(* CODESYS project FsTime_0.1.0.0.library
   Company: FisoThemes
   DefaultNamespace: FsTime
   Version: 0.1.0.0
   Placeholder: FsTime
   Author: Goodwill Mzumala
   Description: A library for time management and manipulation.
   Title: FsTime

Project tree, tasks and I/O mapping:
  libraries: FsCommon, * (FisoThemes); FsError, * (FisoThemes); SysTime, 3.5.9.0 (System); Tc2_Standard, * (Beckhoff Automation GmbH); Tc2_System, * (Beckhoff Automation GmbH); Tc3_Module, * (Beckhoff Automation GmbH)
  DUTs/
    data type E_DayOfWeek
    data type E_Month
    data type E_TimeInstanceKind
    data type T_DayOfMonth
    data type T_DayOfYear
    data type T_Hour
    data type T_Microsecond
    data type T_Millisecond
    data type T_Minute
    data type T_Nanosecond
    data type T_Second
    data type T_Year
  GVLs/
  ITFs/
    Time Instance/
      interface I_ComparableTimesInstance: IsAfter, IsBefore, IsEqualTo
      interface I_EquatableTimesInstance: IsEqualTo
      interface I_TimeInstance: DayOfMonth, DayOfWeek, DayOfYear, EpochMilliseconds, Hour, IsAfter, IsBefore, IsEqualTo, Kind, Millisecond, Minute, Month, Second, ToDate, ToDateTime, ToLocal, ToTimeOfDay, ToUTC, Year
      interface I_TimeInstanceArithmetics
      interface I_TimeInstanceConversions: ToDate, ToDateTime, ToLocal, ToTimeOfDay, ToUTC
      interface I_TimeInstanceProperties: DayOfMonth, DayOfWeek, DayOfYear, EpochMilliseconds, Hour, Kind, Millisecond, Minute, Month, Second, Year
    Time Span/
      interface I_TimeSpan: Day, Hour, Microsecond, Millisecond, Minute, Nanosecond, Second, Tick, ToDays, ToHours, ToMicroseconds, ToMilliseconds, ToMinutes, ToNanoseconds, ToSeconds
      interface I_TimeSpanConversions: ToDays, ToHours, ToMicroseconds, ToMilliseconds, ToMinutes, ToNanoseconds, ToSeconds
      interface I_TimeSpanProperties: Day, Hour, Microsecond, Millisecond, Minute, Nanosecond, Second, Tick
    interface I_IntervalTimer: ElapsedTime, IntervalCount, IntervalTime, IsRunning, Run, SetCallback, Start, Stop
    interface I_Stopwatch: Clear, ElapsedTime, IsRunning, Start, Stop
    interface I_TimeElapsedCallback: OnTimeElapsed
    interface I_Timer: Clear, Duration, ElapsedTime, HasExpired, HasPaused, IsRunning, Pause, Start, Stop, TimeRemaining
    interface I_TimingSource
  POUs/
    function block FB_IntervalTimer [ST]: ElapsedTime, IntervalCount, IntervalTime, IsRunning, Run, SetCallback, Start, Stop
    function block FB_Stopwatch [ST]: Clear, ElapsedTime, IsRunning, Start, Stop
    function block FB_TimeInstance [ST]: DayOfMonth, DayOfWeek, DayOfYear, EpochMilliseconds, FromDate, FromDateTime, FromEpochMilliseconds, FromTime, FromTimeOfDay, Hour, Instance, IsAfter, IsBefore, IsEqualTo, Kind, Millisecond, Minute, Month, Now, Second, ToDate, ToDateTime, ToLocal, ToTimeOfDay, ToUTC, Year
    function block FB_Timer [ST]: Clear, Duration, ElapsedTime, HasExpired, HasPaused, IsRunning, Pause, Start, Stop, TimeRemaining
    function block FB_TimeSpan [ST]: Day, FromShortTime, FromTime, Hour, Microsecond, Millisecond, Minute, Nanosecond, Now, Second, Span, Tick, ToDays, ToHours, ToMicroseconds, ToMilliseconds, ToMinutes, ToNanoseconds, ToSeconds
    program PLAYGROUND [ST]: Example1
  Project Information/
    function F_GetCompany [ST]
    function F_GetTitle [ST]
    function F_GetVersion [ST]
  Version/
    global variables Global_Version
  VISUs/
*)

// DUTs/E_DayOfWeek
// Represents the days of the week.
{attribute 'qualified_only'}
{attribute 'to_string'}
TYPE E_DayOfWeek :
(
	_ := 0, // Uninitialised or default value, representing an undefined day.
	Monday,
	Tuesday,
	Wednesday,
	Thursday,
	Friday,
	Saturday,
	Sunday
) UINT;
END_TYPE

// DUTs/E_Month
// Represents the months of the year.
{attribute 'qualified_only'}
{attribute 'to_string'}
TYPE E_Month :
(
	_ := 0, // Uninitialised or default value, representing an undefined month.
	January,
	February,
	March,
	April,
	May, 
	June, 
	July,
	August,
	September,
	October,
	November,
	December
)UINT;
END_TYPE

// DUTs/E_TimeInstanceKind
{attribute 'qualified_only'}
{attribute 'to_string'}
TYPE E_TimeInstanceKind :
(
	_ := 0, // Uninitialised or default value, indicating an undefined time instance kind.
	UTC,  // The time instance is in Coordinated Universal Time (UTC).
	Local // The time instance is in local time.
);
END_TYPE

// DUTs/T_DayOfMonth
// Represents the day of the current month, with values ranging from 1 to 31, based on the month.
TYPE T_DayOfMonth : UINT(1..31); END_TYPE

// DUTs/T_DayOfYear
// Represents the day of the year, ranging from 1 to 366, where 1 is January 1st,
// and 365 or 366 is December 31st (accounts for leap years).
TYPE T_DayOfYear : UINT(1..366); END_TYPE

// DUTs/T_Hour
// Represents the hours of the current day, based on a 24-hour format, ranging from 0 to 23.
TYPE T_Hour : UINT(0..23); END_TYPE

// DUTs/T_Microsecond
// Represents the microseconds of the current millisecond, ranging from 0 to 999.
TYPE T_Microsecond : UINT(0..999); END_TYPE

// DUTs/T_Millisecond
// Represents the milliseconds of the current second, ranging from 0 to 999.
TYPE T_Millisecond : UINT(0..999); END_TYPE

// DUTs/T_Minute
// Represents the minutes of the current hour, ranging from 0 to 59.
TYPE T_Minute : UINT(0..59); END_TYPE

// DUTs/T_Nanosecond
// Represents the nanoseconds of the current microsecond, ranging from 0 to 999.
TYPE T_Nanosecond : UINT(0..999); END_TYPE

// DUTs/T_Second
// Represents the seconds of the current minute, ranging from 0 to 59.
TYPE T_Second : UINT(0..59); END_TYPE

// DUTs/T_Year
// Represents the year as a four-digit value (e.g., 2024).
TYPE T_Year : UINT; END_TYPE

// Version/Global_Version
{attribute 'TcGenerated'}
{attribute 'no-analysis'}
{attribute 'linkalways'}
// This function has been automatically generated from the project information.
VAR_GLOBAL CONSTANT
	{attribute 'const_non_replaced'}
	stLibVersion_FsTime : ST_LibVersion := (iMajor := 0, iMinor := 1, iBuild := 0, iRevision := 0, nFlags := 0, sVersion := '0.1.0.0');
END_VAR

// ITFs/Time Instance/I_ComparableTimesInstance
// This interface defines operations for comparing time instance objects within a system.
INTERFACE I_ComparableTimesInstance EXTENDS __SYSTEM.IQueryInterface

// Checks if the current time instance is after the specified time instance.
METHOD IsAfter : BOOL // TRUE if the current time instance is after the specified one, FALSE otherwise.
VAR_INPUT
	// The time instance to compare against.
	ipOther : I_TimeInstance;
END_VAR
END_METHOD

// Checks if the current time instance is before the specified time instance.
METHOD IsBefore : BOOL // TRUE if the current time instance is before the specified one, FALSE otherwise.
VAR_INPUT
	// The time instance to compare against.
	ipOther : I_TimeInstance;
END_VAR
END_METHOD

// Checks if the current time instance is equal to the specified time instance.
METHOD IsEqualTo : BOOL // TRUE if the current time instance is equal to the specified, FALSE otherwise.
VAR_INPUT
	// The time instance to compare against.
	ipOther : I_TimeInstance;
END_VAR
END_METHOD

END_INTERFACE

// ITFs/Time Instance/I_TimeInstance
// Interface for a time instance.
INTERFACE I_TimeInstance EXTENDS __SYSTEM.IQueryInterface

// The day of the month extracted from the time instance.
// [get] Returns the day component of the date, with a value ranging from 1 to 31.
PROPERTY DayOfMonth : T_DayOfMonth
GET
END_GET
END_PROPERTY

// The day of the week extracted from the time instance.
// [get] Returns the day as an `E_DayOfWeek` enum or value ranging from 1 (Monday) to 7 (Sunday).
PROPERTY DayOfWeek : E_DayOfWeek
GET
END_GET
END_PROPERTY

// The day of the year extracted from the time instance.
// [get] Returns the day of the year, with a value ranging from 1 to 366.
PROPERTY DayOfYear : T_DayOfYear
GET
END_GET
END_PROPERTY

// The time instance value represented as the number of milliseconds since
// Thursday, 1.1.1970 00:00:00.000 (Unix epoch).
// [get] Returns the time instance value in milliseconds.
PROPERTY EpochMilliseconds : ULINT
GET
END_GET
END_PROPERTY

// The hour of the day extracted from the time instance.
// [get] Returns the hour component of the time, with a value ranging from 0 to 23.
PROPERTY Hour : T_Hour
GET
END_GET
END_PROPERTY

// Checks if the current time instance is after the specified time instance.
METHOD IsAfter : BOOL // TRUE if the current time instance is after the specified one, FALSE otherwise.
VAR_INPUT
	// The time instance to compare against.
	ipOther : I_TimeInstance;
END_VAR
END_METHOD

// Checks if the current time instance is before the specified time instance.
METHOD IsBefore : BOOL // TRUE if the current time instance is before the specified one, FALSE otherwise.
VAR_INPUT
	// The time instance to compare against.
	ipOther : I_TimeInstance;
END_VAR
END_METHOD

// Checks if the current time instance is equal to the specified time instance.
METHOD IsEqualTo : BOOL // TRUE if the current time instance is equal to the specified, FALSE otherwise.
VAR_INPUT
	// The time instance to compare against.
	ipOther : I_TimeInstance;
END_VAR
END_METHOD

// Specifies whether the time instance is in UTC or local time format.
// [get] Returns the time instance type enum as a value.
PROPERTY Kind : E_TimeInstanceKind
GET
END_GET
END_PROPERTY

// The millisecond part of the second extracted from the time instance.
// [get] Returns the millisecond component, with a value ranging from 0 to 999.
PROPERTY Millisecond : T_Millisecond
GET
END_GET
END_PROPERTY

// The minute of the hour extracted from the time instance.
// [get] Returns the minute component, with a value ranging from 0 to 59.
PROPERTY Minute : T_Minute
GET
END_GET
END_PROPERTY

// The month of the year extracted from the time instance.
// [get] Returns the month as an `E_Month` enum or a value ranging from 1 to 12 value.
PROPERTY Month : E_Month
GET
END_GET
END_PROPERTY

// The second of the minute extracted from the time instance.
// [get] Returns the second component, with a value ranging from 0 to 59.
PROPERTY Second : T_Second
GET
END_GET
END_PROPERTY

// Converts the time instance to a date value.
METHOD ToDate : DATE // The date part of the time instance.
VAR_OUTPUT
	// Error code indicating the result of the operation.
	Error : FsError.T_Error;
END_VAR
END_METHOD

// Converts the time instance to a combined date and time value.
METHOD ToDateTime : DT // The combined date and time value as a DT (Date and Time).
VAR_OUTPUT
	// Error code indicating the result of the operation.
	Error : FsError.T_Error;
END_VAR
END_METHOD

// Converts the time instance to local time representation.
METHOD ToLocal : I_TimeInstance // A reference to the current instance.
VAR_OUTPUT
	// Error code indicating the result of the operation.
	Error : FsError.T_Error;
END_VAR
END_METHOD

// Converts the time instance to a time of day  value.
METHOD ToTimeOfDay : TOD // The time of day part of the time instance.
VAR_INPUT
END_VAR
END_METHOD

// Converts the time instance to UTC time representation.
METHOD ToUTC : I_TimeInstance // A reference to the current instance.
VAR_OUTPUT
	// Error code indicating the result of the operation.
	Error : FsError.T_Error;
END_VAR
END_METHOD

// The year extracted from the time instance.
// [get] Returns the year as a 4 digit value.
PROPERTY Year : T_Year
GET
END_GET
END_PROPERTY

END_INTERFACE

// ITFs/Time Instance/I_EquatableTimesInstance
// This interface defines the operations for equality between time instance objects within a system.
INTERFACE I_EquatableTimesInstance EXTENDS __SYSTEM.IQueryInterface

// Checks if the current time instance is equal to the specified time instance.
METHOD IsEqualTo : BOOL // TRUE if the current time instance is equal to the specified, FALSE otherwise.
VAR_INPUT
	// The time instance to compare against.
	ipOther : I_TimeInstance;
END_VAR
END_METHOD

END_INTERFACE

// ITFs/Time Instance/I_TimeInstanceArithmetics
// Interface that defines the arithmetic operations for a time instance.
INTERFACE I_TimeInstanceArithmetics EXTENDS __SYSTEM.IQueryInterface

END_INTERFACE

// ITFs/Time Instance/I_TimeInstanceConversions
// Interface that defines operations for converting a time instance to different representations.
INTERFACE I_TimeInstanceConversions EXTENDS __SYSTEM.IQueryInterface

// Converts the time instance to a date value.
METHOD ToDate : DATE // The date part of the time instance.
VAR_OUTPUT
	// Error code indicating the result of the operation.
	Error : FsError.T_Error;
END_VAR
END_METHOD

// Converts the time instance to a combined date and time value.
METHOD ToDateTime : DT // The combined date and time value as a DT (Date and Time).
VAR_OUTPUT
	// Error code indicating the result of the operation.
	Error : FsError.T_Error;
END_VAR
END_METHOD

// Converts the time instance to local time representation.
METHOD ToLocal : I_TimeInstance // A reference to the current instance.
VAR_OUTPUT
	// Error code indicating the result of the operation.
	Error : FsError.T_Error;
END_VAR
END_METHOD

// Converts the time instance to a time of day  value.
METHOD ToTimeOfDay : TOD // The time of day part of the time instance.
VAR_INPUT
END_VAR
END_METHOD

// Converts the time instance to UTC time representation.
METHOD ToUTC : I_TimeInstance // A reference to the current instance.
VAR_OUTPUT
	// Error code indicating the result of the operation.
	Error : FsError.T_Error;
END_VAR
END_METHOD

END_INTERFACE

// ITFs/Time Instance/I_TimeInstanceProperties
// Inertface for defining the basic properties of a time instance.
INTERFACE I_TimeInstanceProperties EXTENDS __SYSTEM.IQueryInterface

// The day of the month extracted from the time instance.
// [get] Returns the day component of the date, with a value ranging from 1 to 31.
PROPERTY DayOfMonth : T_DayOfMonth
GET
END_GET
END_PROPERTY

// The day of the week extracted from the time instance.
// [get] Returns the day as an `E_DayOfWeek` enum or value ranging from 1 (Monday) to 7 (Sunday).
PROPERTY DayOfWeek : E_DayOfWeek
GET
END_GET
END_PROPERTY

// The day of the year extracted from the time instance.
// [get] Returns the day of the year, with a value ranging from 1 to 366.
PROPERTY DayOfYear : T_DayOfYear
GET
END_GET
END_PROPERTY

// The time instance value represented as the number of milliseconds since
// Thursday, 1.1.1970 00:00:00.000 (Unix epoch).
// [get] Returns the time instance value in milliseconds.
PROPERTY EpochMilliseconds : ULINT
GET
END_GET
END_PROPERTY

// The hour of the day extracted from the time instance.
// [get] Returns the hour component of the time, with a value ranging from 0 to 23.
PROPERTY Hour : T_Hour
GET
END_GET
END_PROPERTY

// Specifies whether the time instance is in UTC or local time format.
// [get] Returns the time instance type enum as a value.
PROPERTY Kind : E_TimeInstanceKind
GET
END_GET
END_PROPERTY

// The millisecond part of the second extracted from the time instance.
// [get] Returns the millisecond component, with a value ranging from 0 to 999.
PROPERTY Millisecond : T_Millisecond
GET
END_GET
END_PROPERTY

// The minute of the hour extracted from the time instance.
// [get] Returns the minute component, with a value ranging from 0 to 59.
PROPERTY Minute : T_Minute
GET
END_GET
END_PROPERTY

// The month of the year extracted from the time instance.
// [get] Returns the month as an `E_Month` enum or a value ranging from 1 to 12 value.
PROPERTY Month : E_Month
GET
END_GET
END_PROPERTY

// The second of the minute extracted from the time instance.
// [get] Returns the second component, with a value ranging from 0 to 59.
PROPERTY Second : T_Second
GET
END_GET
END_PROPERTY

// The year extracted from the time instance.
// [get] Returns the year as a 4 digit value.
PROPERTY Year : T_Year
GET
END_GET
END_PROPERTY

END_INTERFACE

// ITFs/Time Span/I_TimeSpan
INTERFACE I_TimeSpan EXTENDS __SYSTEM.IQueryInterface

// The day component of the time span.
// [get] Returns the day component of the time, with a value ranging from 0 to 213503.
PROPERTY Day : UDINT(0..213503)
GET
END_GET
END_PROPERTY

// The hour component of the time span.
// [get] Returns the hour component of the time, with a value ranging from 0 to 23.
PROPERTY Hour : T_Hour
GET
END_GET
END_PROPERTY

// The microsecond component of the time span.
// [get] Returns the microsecond component, with a value ranging from 0 to 999.
PROPERTY Microsecond : T_Microsecond
GET
END_GET
END_PROPERTY

// The millisecond component of the time span.
// [get] Returns the millisecond component, with a value ranging from 0 to 999.
PROPERTY Millisecond : T_Millisecond
GET
END_GET
END_PROPERTY

// The minute component of the time span.
// [get] Returns the minute component, with a value ranging from 0 to 59.
PROPERTY Minute : T_Minute
GET
END_GET
END_PROPERTY

// The nanosecond component of the time span.
// [get] Returns the nanosecond component, with a value ranging from 0 to 999.
PROPERTY Nanosecond : T_Nanosecond
GET
END_GET
END_PROPERTY

// The second component of the time span.
// [get] Returns the second component, with a value ranging from 0 to 59.
PROPERTY Second : T_Second
GET
END_GET
END_PROPERTY

// Represents the time span as LTIME.
// [get] Returns the time span value as an LTIME, which can be used for time calculations and comparisons.
PROPERTY Tick : LTIME
GET
END_GET
END_PROPERTY

// Converts the time span represented by the instance into days.
METHOD ToDays : ULINT // The total number of days in the time span.
VAR_INPUT
END_VAR
END_METHOD

// Converts the time span represented by the instance into hours.
METHOD ToHours : ULINT // The total number of hours in the time span.
VAR_INPUT
END_VAR
END_METHOD

// Converts the time span represented by the instance into microseconds.
METHOD ToMicroseconds : ULINT // The total number of microseconds in the time span.
VAR_INPUT
END_VAR
END_METHOD

// Converts the time span represented by the instance into milliseconds.
METHOD ToMilliseconds : ULINT // The total number of milliseconds in the time span.
VAR_INPUT
END_VAR
END_METHOD

// Converts the time span represented by the instance into minutes.
METHOD ToMinutes : ULINT // The total number of minutes in the time span.
VAR_INPUT
END_VAR
END_METHOD

// Converts the time span represented by the instance into nanoseconds.
METHOD ToNanoseconds : ULINT // The total number of nanoseconds in the time span.
VAR_INPUT
END_VAR
END_METHOD

// Converts the time span represented by the instance into seconds.
METHOD ToSeconds : ULINT // The total number of seconds in the time span.
VAR_INPUT
END_VAR
END_METHOD

END_INTERFACE

// ITFs/Time Span/I_TimeSpanConversions
INTERFACE I_TimeSpanConversions

// Converts the time span represented by the instance into days.
METHOD ToDays : ULINT // The total number of days in the time span.
VAR_INPUT
END_VAR
END_METHOD

// Converts the time span represented by the instance into hours.
METHOD ToHours : ULINT // The total number of hours in the time span.
VAR_INPUT
END_VAR
END_METHOD

// Converts the time span represented by the instance into microseconds.
METHOD ToMicroseconds : ULINT // The total number of microseconds in the time span.
VAR_INPUT
END_VAR
END_METHOD

// Converts the time span represented by the instance into milliseconds.
METHOD ToMilliseconds : ULINT // The total number of milliseconds in the time span.
VAR_INPUT
END_VAR
END_METHOD

// Converts the time span represented by the instance into minutes.
METHOD ToMinutes : ULINT // The total number of minutes in the time span.
VAR_INPUT
END_VAR
END_METHOD

// Converts the time span represented by the instance into nanoseconds.
METHOD ToNanoseconds : ULINT // The total number of nanoseconds in the time span.
VAR_INPUT
END_VAR
END_METHOD

// Converts the time span represented by the instance into seconds.
METHOD ToSeconds : ULINT // The total number of seconds in the time span.
VAR_INPUT
END_VAR
END_METHOD

END_INTERFACE

// ITFs/Time Span/I_TimeSpanProperties
INTERFACE I_TimeSpanProperties

// The day component of the time span.
// [get] Returns the day component of the time, with a value ranging from 0 to 213503.
PROPERTY Day : UDINT(0..213503)
GET
END_GET
END_PROPERTY

// The hour component of the time span.
// [get] Returns the hour component of the time, with a value ranging from 0 to 23.
PROPERTY Hour : T_Hour
GET
END_GET
END_PROPERTY

// The microsecond component of the time span.
// [get] Returns the microsecond component, with a value ranging from 0 to 999.
PROPERTY Microsecond : T_Microsecond
GET
END_GET
END_PROPERTY

// The millisecond component of the time span.
// [get] Returns the millisecond component, with a value ranging from 0 to 999.
PROPERTY Millisecond : T_Millisecond
GET
END_GET
END_PROPERTY

// The minute component of the time span.
// [get] Returns the minute component, with a value ranging from 0 to 59.
PROPERTY Minute : T_Minute
GET
END_GET
END_PROPERTY

// The nanosecond component of the time span.
// [get] Returns the nanosecond component, with a value ranging from 0 to 999.
PROPERTY Nanosecond : T_Nanosecond
GET
END_GET
END_PROPERTY

// The second component of the time span.
// [get] Returns the second component, with a value ranging from 0 to 59.
PROPERTY Second : T_Second
GET
END_GET
END_PROPERTY

// Represents the time span as LTIME.
// [get] Returns the time span value as an LTIME, which can be used for time calculations and comparisons.
PROPERTY Tick : LTIME
GET
END_GET
END_PROPERTY

END_INTERFACE

// ITFs/I_IntervalTimer
// This interface defines the behaviour of an interval timer, a type of timing source
// that operates based on a specified interval. It is intended to be used for periodic
// actions or repeated timing events.
INTERFACE I_IntervalTimer EXTENDS I_TimingSource

// The elapsed time since the timer was started or last reset, showing how much time has passed within the current interval.
// [get] Returns the elapsed time within the current interval.
PROPERTY ElapsedTime  : LTIME
GET
END_GET
END_PROPERTY

// The number of intervals that have elapsed since the timer was started or reset.
// [get] Returns the number of elapsed intervals.
PROPERTY IntervalCount : FsCommon.T_Size
GET
END_GET
END_PROPERTY

// The interval duration for the timer. It specifies how long the timer should wait between triggers.
// [get] Returns the interval duration.
// [set] Sets the interval duration.
PROPERTY IntervalTime : LTIME
GET
END_GET
SET
END_SET
END_PROPERTY

// Indicates whether the interval timer is currently running.
// [get] Returns TRUE if the timer is running; otherwise, FALSE.
PROPERTY IsRunning  : BOOL
GET
END_GET
END_PROPERTY

// The method that must be called cyclically to run the interval timer.
METHOD Run : I_IntervalTimer // Reference to the current instance of I_IntervalTimer.
VAR_INPUT
END_VAR
END_METHOD

// Sets the callback to be invoked when the interval has elapsed.
METHOD SetCallback : I_IntervalTimer // Reference to the current instance of I_IntervalTimer.
VAR_INPUT
	// The callback that is invoked when the interval elapses.
    ipCallback : I_TimeElapsedCallback;
END_VAR
END_METHOD

// Starts the interval timer, beginning the measurement of time intervals.
METHOD Start : I_IntervalTimer // Reference to the current instance of I_IntervalTimer.
VAR_INPUT
END_VAR
END_METHOD

// Stops the interval timer, halting the measurement of time intervals.
METHOD Stop : I_IntervalTimer // Reference to the current instance of I_IntervalTimer.
VAR_INPUT
END_VAR
END_METHOD

END_INTERFACE

// ITFs/I_TimingSource
// This interface serves as a marker or base type for various timing sources.
// It allows for the use of polymorphism and type checking when working with
// different timing sources, such as timers, stopwatches, and interval timers.
INTERFACE I_TimingSource EXTENDS __SYSTEM.IQueryInterface

END_INTERFACE

// ITFs/I_TimeElapsedCallback
// This interface is designed to be implemented by objects that need to respond
// to time elapsed events from timing sources such as timers or interval timers.
INTERFACE I_TimeElapsedCallback EXTENDS __SYSTEM.IQueryInterface

// This method is called when the associated timing source reaches the elapsed time
// threshold. Implementers should define the specific actions to be taken when
// this event occurs.
METHOD OnTimeElapsed
VAR_INPUT
    // An instance of the timing source representing the source of the elapsed time event.
    // This instance can be queried for its specific type using the __QUERYINTERFACE
    // function, allowing for tailored handling based on the source's type.
	ipSource : I_TimingSource;
END_VAR
END_METHOD

END_INTERFACE

// ITFs/I_Stopwatch
// This interface defines the behaviour of a stopwatch, a type of timing source 
// used to measure the elapsed time between the start and stop actions. It can
// be cleared to reset the elapsed time and is useful for timing events,
// measuring durations, or performance monitoring.
INTERFACE I_Stopwatch EXTENDS I_TimingSource

// Clears the stopwatch, resetting the elapsed time to zero.
METHOD Clear
VAR_INPUT
END_VAR
END_METHOD

// The elapsed time measured by the stopwatch since it was started.
// [get] Returns the elapsed time.
PROPERTY ElapsedTime  : LTIME
GET
END_GET
END_PROPERTY

// Indicates whether the stopwatch is currently running.
// [get] Returns TRUE if the stopwatch is running; otherwise, FALSE.
PROPERTY IsRunning  : BOOL
GET
END_GET
END_PROPERTY

// Starts the stopwatch, beginning the measurement of elapsed time.
METHOD Start
VAR_INPUT
END_VAR
END_METHOD

// Stops the stopwatch, halting the measurement of elapsed time.
METHOD Stop
VAR_INPUT
END_VAR
END_METHOD

END_INTERFACE

// ITFs/I_Timer
// This interface defines the behaviour of a timer, a type of timing source used
// to track a specific duration. The timer can be started, paused, stopped, and
// cleared. It is commonly used for timing events, delays, and other time-based
// operations. The timer tracks elapsed time and can indicate when the set 
// duration has expired.
INTERFACE I_Timer EXTENDS I_TimingSource

// Clears the timer, resetting the elapsed time.
METHOD Clear
VAR_INPUT
END_VAR
END_METHOD

// The duration for the timer. It specifies how long the timer should run before
// it expires.
// [get] Returns the set duration.
// [set] Sets the duration for the timer.
PROPERTY Duration : LTIME
GET
END_GET
SET
END_SET
END_PROPERTY

// The elapsed time since the timer was started.
// [get] Returns the elapsed time.
PROPERTY ElapsedTime  : LTIME
GET
END_GET
END_PROPERTY

// Indicates whether the timer has expired.
// [get] Returns TRUE if the timer has expired; otherwise, FALSE.
PROPERTY HasExpired : BOOL
GET
END_GET
END_PROPERTY

// Indicates whether the timer is currently paused.
// [get] Returns TRUE if the timer is paused; otherwise, FALSE.
PROPERTY HasPaused : BOOL
GET
END_GET
END_PROPERTY

// Indicates whether the timer is currently running.
// [get] Returns TRUE if the timer is running; otherwise, FALSE.
PROPERTY IsRunning  : BOOL
GET
END_GET
END_PROPERTY

// Pauses the timer, preserving the elapsed time without resetting.
METHOD Pause
VAR_INPUT
END_VAR
END_METHOD

// Starts the timer, beginning the tracking of time towards the specified duration.
METHOD Start
VAR_INPUT
END_VAR
END_METHOD

// Stops the timer, halting the tracking of time.
METHOD Stop
VAR_INPUT
END_VAR
END_METHOD

// The remaining time until the timer expires.
// [get] Returns the time remaining until expiration.
PROPERTY TimeRemaining : LTIME
GET
END_GET
END_PROPERTY

END_INTERFACE

// POUs/FB_IntervalTimer
// A timer that triggers at regular intervals. It tracks elapsed time in
// nanoseconds and invokes a user-defined callback when each interval is reached.
// This block is particularly useful in scenarios where repeated actions are
// needed at precise time intervals, such as generating periodic events or
// monitoring cyclic processes.
//
// [usage] 
// The timer can be started with the `Start` method, and the `Run` method should
// be called within a cyclic task to continuously update the timer state. The
// `IntervalCount` property can be used to specify the duration between triggers, and
// the callback method will be called each time this duration is met.
{attribute 'enable_dynamic_creation'}
{attribute 'no_explicit_call' := 'direct call for this function block is not allowed'}
FUNCTION_BLOCK FINAL FB_IntervalTimer IMPLEMENTS I_IntervalTimer
VAR
	_tIntervalTime	: LTIME; // Duration between each interval trigger.
	_tTick			: LTIME; // Timestamp at which the timer was last started or reset.
	_tElapsedTime 	: LTIME; // Total elapsed time since the timer was started.
	_bIsRunning 	: BOOL;  // Indicating whether the interval timer is currently running.
	_IntervalCount 	: FsCommon.T_Size; // Number of intervals that have passed since the timer started.
	_ipCallback 	: I_TimeElapsedCallback; // Reference to the callback that will be invoked when the interval is reached.
END_VAR

// The elapsed time since the timer was started or last reset, showing how much time has passed within the current interval.
// [get] Returns the elapsed time within the current interval.
PROPERTY ElapsedTime  : LTIME
GET
ElapsedTime := THIS^._tElapsedTime;
END_GET
END_PROPERTY

// The number of intervals that have elapsed since the timer was started or reset.
// [get] Returns the number of elapsed intervals.
PROPERTY IntervalCount : FsCommon.T_Size
GET
IntervalCount := THIS^._IntervalCount;
END_GET
END_PROPERTY

// The interval duration for the timer. It specifies how long the timer should wait between triggers.
// [get] Returns the interval duration.
// [set] Sets the interval duration.
PROPERTY IntervalTime : LTIME
GET
IntervalTime := THIS^._tIntervalTime;
END_GET
SET
THIS^._tIntervalTime := IntervalTime;
END_SET
END_PROPERTY

// Indicates whether the interval timer is currently running.
// [get] Returns TRUE if the timer is running; otherwise, FALSE.
PROPERTY IsRunning  : BOOL
GET
IsRunning := THIS^._bIsRunning;
END_GET
END_PROPERTY

// The method that must be called cyclically to run the interval timer.
METHOD Run : I_IntervalTimer // Reference to the current instance of I_IntervalTimer.
VAR_INPUT
END_VAR
Run := THIS^;

IF NOT THIS^._bIsRunning THEN RETURN; END_IF

THIS^._tElapsedTime := LTIME() - THIS^._tTick;

IF THIS^._tElapsedTime < THIS^._tIntervalTime THEN RETURN; END_IF

THIS^._IntervalCount := THIS^._IntervalCount + 1;
IF THIS^._ipCallback <> 0 THEN THIS^._ipCallback.OnTimeElapsed(THIS^); END_IF
THIS^._tTick := LTIME();
END_METHOD

// Sets the callback to be invoked when the interval has elapsed.
METHOD SetCallback : I_IntervalTimer // Reference to the current instance of I_IntervalTimer.
VAR_INPUT
	// The callback that is invoked when the interval elapses.
    ipCallback : I_TimeElapsedCallback;
END_VAR
THIS^._ipCallback := ipCallback;
END_METHOD

// Starts the interval timer, beginning the measurement of time intervals.
METHOD Start : I_IntervalTimer // Reference to the current instance of I_IntervalTimer.
VAR_INPUT
END_VAR
Start := THIS^;

IF THIS^._bIsRunning THEN RETURN; END_IF

THIS^._tElapsedTime 	:= LTIME#0S;
THIS^._IntervalCount 	:= 0;
THIS^._tTick 			:= LTIME();
THIS^._bIsRunning 		:= TRUE;
END_METHOD

// Stops the interval timer, halting the measurement of time intervals.
METHOD Stop : I_IntervalTimer // Reference to the current instance of I_IntervalTimer.
VAR_INPUT
END_VAR
Stop := THIS^;

THIS^._bIsRunning := FALSE;
END_METHOD

END_FUNCTION_BLOCK

// POUs/FB_Stopwatch
// A simple stopwatch that tracks elapsed time between a start and stop event.
// The stopwatch can be cleared to reset the elapsed time.
//
// [usage]
// Call the `Start` method to begin timing. The `ElapsedTime` property will track
// the time until the `Stop` method is called. To reset the elapsed time, use the
// `Clear` method.
{attribute 'enable_dynamic_creation'}
{attribute 'no_explicit_call' := 'direct call for this function block is not allowed'}
FUNCTION_BLOCK FINAL FB_Stopwatch IMPLEMENTS I_Stopwatch
VAR
    _tStartTime     : LTIME; // Timestamp when the stopwatch was started.
    _tElapsedTime   : LTIME; // Accumulated elapsed time.
    _bIsRunning     : BOOL;  // Indicates if the stopwatch is currently running.
END_VAR

// Clears the stopwatch, resetting the elapsed time to zero.
METHOD Clear
VAR_INPUT
END_VAR
THIS^._tElapsedTime := LTIME#0S;
IF THIS^._bIsRunning THEN THIS^._tStartTime := LTIME(); END_IF
END_METHOD

// The elapsed time measured by the stopwatch since it was started.
// [get] Returns the elapsed time.
PROPERTY ElapsedTime  : LTIME
GET
ElapsedTime := THIS^._tElapsedTime := 
	SEL(
		THIS^._bIsRunning,
		THIS^._tElapsedTime,
		LTIME() - THIS^._tStartTime);
END_GET
END_PROPERTY

// Indicates whether the stopwatch is currently running.
// [get] Returns TRUE if the stopwatch is running; otherwise, FALSE.
PROPERTY IsRunning  : BOOL
GET
IsRunning := THIS^._bIsRunning;
END_GET
END_PROPERTY

// Starts the stopwatch, beginning the measurement of elapsed time.
METHOD Start
VAR_INPUT
END_VAR
IF THIS^._bIsRunning THEN RETURN; END_IF

THIS^._tStartTime := LTIME();
THIS^._bIsRunning := TRUE;
END_METHOD

// Stops the stopwatch, halting the measurement of elapsed time.
METHOD Stop
VAR_INPUT
END_VAR
IF NOT THIS^._bIsRunning THEN RETURN; END_IF

THIS^._tElapsedTime := THIS^._tElapsedTime := LTIME() - THIS^._tStartTime;
THIS^._bIsRunning 	:= FALSE;
END_METHOD

END_FUNCTION_BLOCK

// POUs/FB_TimeInstance
// A time instance function block that represents a date and time value based on the Unix epoch (1st Jan 1970, 00:00:00.000).
// The block provides various methods and properties to interact with the time instance, including support for UTC and local time representations.
// It can be used for time calculations, comparisons, and conversions to different time formats (e.g., `DT`, `DATE`, `TOD`).
//
// [usage]
// The time instance can be set using various methods such as `FromDateTime` or `FromEpochMilliseconds`. 
// Use properties like `Year`, `Month`, `DayOfMonth`, `Hour`, and `Minute` to extract specific components of the date and time.
// Additionally, the `ToLocal` and `ToUTC` properties allow switching between different time modes.
// Use the `Kind` property to check the time mode.
{attribute 'enable_dynamic_creation'}
{attribute 'no_explicit_call' := 'calling this function block directly is not allowed'}
FUNCTION_BLOCK FINAL FB_TimeInstance 
IMPLEMENTS 
	I_TimeInstance, I_ComparableTimesInstance, I_EquatableTimesInstance, 
	I_TimeInstanceProperties, I_TimeInstanceArithmetics, I_TimeInstanceConversions
VAR
    _nEpochMilliseconds : ULINT; // The raw time instance value in milliseconds since 1st Jan 1970.
    _Date				: SysTimeRtc.SYSTIMEDATE; // Structured representation of the time instance (year, month, day, etc.).
    _eKind				: E_TimeInstanceKind; // Indicates whether the time instance is in UTC or Local time.
END_VAR

// The day of the month extracted from the time instance.
// [get] Returns the day component of the date, with a value ranging from 1 to 31.
PROPERTY DayOfMonth : T_DayOfMonth
GET
DayOfMonth := THIS^._Date.wDay;
END_GET
END_PROPERTY

// The day of the week extracted from the time instance.
// [get] Returns the day as an `E_DayOfWeek` enum or value ranging from 1 (Monday) to 7 (Sunday).
PROPERTY DayOfWeek : E_DayOfWeek
GET
DayOfWeek := THIS^._Date.wDayOfWeek;
END_GET
END_PROPERTY

// The day of the year extracted from the time instance.
// [get] Returns the day of the year, with a value ranging from 1 to 366.
PROPERTY DayOfYear : T_DayOfYear
GET
DayOfYear := THIS^._Date.wYday;
END_GET
END_PROPERTY

// The time instance value represented as the number of milliseconds since
// Thursday, 1.1.1970 00:00:00.000 (Unix epoch).
// [get] Returns the time instance value in milliseconds.
PROPERTY EpochMilliseconds : ULINT
GET
EpochMilliseconds := THIS^._nEpochMilliseconds;
END_GET
END_PROPERTY

// Sets the time instance based on a given `DATE` value as UTC.
METHOD FromDate : I_TimeInstance // A reference to the current instance.
VAR_INPUT
	// The input `DATE` value to convert to a time instance.
	dValue : DATE;
END_VAR
VAR_OUTPUT
	// Error code indicating the result of the operation.
	Error : FsError.T_Error;
END_VAR
FromDate := THIS^;

THIS^.FromEpochMilliseconds(TO_ULINT(dValue) * 1000, Error => Error);
END_METHOD

// Sets the time instance based on a given `DT` (Date and Time) value as UTC.
METHOD FromDateTime : I_TimeInstance // A reference to the current instance.
VAR_INPUT
	// The input `DT` value to convert to a time instance.
	dtValue : DT;
END_VAR
VAR_OUTPUT
	// Error code indicating the result of the operation.
	Error : FsError.T_Error;
END_VAR
FromDateTime := THIS^;

THIS^.FromEpochMilliseconds(TO_ULINT(dtValue) * 1000, Error => Error);
END_METHOD

// Sets the time instance based on a given number of milliseconds since the Unix epoch (1st Jan 1970, 00:00:00.000).
METHOD FromEpochMilliseconds : I_TimeInstance // A reference to the current instance.
VAR_INPUT
	// The input time instance value representing the number of milliseconds since 1st Jan 1970, 00:00:00.000.
	nValue : ULINT;
END_VAR
VAR_OUTPUT
	// Error code indicating the result of the operation.
	Error : FsError.T_Error;
END_VAR
VAR
	eResult : FsError.E_CodesysCmpError;
END_VAR
FromEpochMilliseconds := THIS^;

IF THIS^._nEpochMilliseconds = nValue THEN RETURN; END_IF

eResult := SysTimeRtc.SysTimeRtcConvertHighResToDate(nValue, THIS^._Date);
CASE eResult OF
	FsError.E_CodesysCmpError.ERR_OK:
		THIS^._eKind := E_TimeInstanceKind.UTC;
		THIS^._nEpochMilliseconds := nValue;
ELSE
	Error := 
		FsError.F_CreateErrorFromStartRange(
			FsError.GVL_ErrorDescriptors.fbGeneralErrorCodes,
			FsError.E_GeneralErrorCode.ERR_CODESYS_BEGIN,
			eResult);
	THIS^.FB_init(FALSE, FALSE);
	END_CASE
END_METHOD

// Sets the time instance using the specified `LTIME` value. 
// This method converts the input value to milliseconds since the Unix epoch (1st Jan 1970, 00:00:00.000). 
//
// [note] 
// The method only considers the time value down to the millisecond precision. 
// Any values smaller than 1ms (e.g., microseconds or nanoseconds) will be ignored.
METHOD FromTime : I_TimeInstance // A reference to the current instance.
VAR_INPUT
	// The time value to be set, provided as an LTIME datatype (milliseconds since the Unix epoch).
	tValue : LTIME;
END_VAR
VAR_OUTPUT
	// Error code indicating the result of the operation.
	Error : FsError.T_Error;
END_VAR
FromTime := THIS^;

THIS^.FromEpochMilliseconds(TO_ULINT(tValue) / TO_ULINT(LTIME#1MS), Error => Error);
END_METHOD

// Sets the time instance based on a given `TOD` (Time Of Day) value as UTC.
METHOD FromTimeOfDay : I_TimeInstance // A reference to the current instance.
VAR_INPUT
	// The input `TOD` value to convert to a time instance.
	tdValue : TOD;
END_VAR
VAR_OUTPUT
	// Error code indicating the result of the operation.
	Error : FsError.T_Error;
END_VAR
FromTimeOfDay := THIS^;

THIS^.FromEpochMilliseconds(TO_ULINT(tdValue), Error => Error);
END_METHOD

// The hour of the day extracted from the time instance.
// [get] Returns the hour component of the time, with a value ranging from 0 to 23.
PROPERTY Hour : T_Hour
GET
Hour := THIS^._Date.wHour;
END_GET
END_PROPERTY

// The reference to the current time instance.
// [get] Returns a reference to the current time instance implementing `I_TimeInstance`.
PROPERTY Instance : I_TimeInstance
GET
Instance := THIS^;
END_GET
END_PROPERTY

// Checks if the current time instance is after the specified time instance.
METHOD IsAfter : BOOL // TRUE if the current time instance is after the specified one, FALSE otherwise.
VAR_INPUT
	// The time instance to compare against.
	ipOther : I_TimeInstance;
END_VAR
IsAfter := 
	ipOther <> 0
	AND_THEN
	THIS^._nEpochMilliseconds > ipOther.EpochMilliseconds;
END_METHOD

// Checks if the current time instance is before the specified time instance.
METHOD IsBefore : BOOL // TRUE if the current time instance is before the specified one, FALSE otherwise.
VAR_INPUT
	// The time instance to compare against.
	ipOther : I_TimeInstance;
END_VAR
IsBefore := 
	ipOther <> 0
	AND_THEN
	THIS^._nEpochMilliseconds < ipOther.EpochMilliseconds;
END_METHOD

// Checks if the current time instance is equal to the specified time instance.
METHOD IsEqualTo : BOOL // TRUE if the current time instance is equal to the specified, FALSE otherwise.
VAR_INPUT
	// The time instance to compare against.
	ipOther : I_TimeInstance;
END_VAR
IsEqualTo := 
	ipOther <> 0
	AND_THEN
	THIS^._nEpochMilliseconds = ipOther.EpochMilliseconds;
END_METHOD

// Specifies whether the time instance is in UTC or local time format.
// [get] Returns the time instance type enum as a value.
PROPERTY Kind : E_TimeInstanceKind
GET
Kind := THIS^._eKind;
END_GET
END_PROPERTY

// The millisecond part of the second extracted from the time instance.
// [get] Returns the millisecond component, with a value ranging from 0 to 999.
PROPERTY Millisecond : T_Millisecond
GET
Millisecond := THIS^._Date.wMilliseconds;
END_GET
END_PROPERTY

// The minute of the hour extracted from the time instance.
// [get] Returns the minute component, with a value ranging from 0 to 59.
PROPERTY Minute : T_Minute
GET
Minute := THIS^._Date.wMinute;
END_GET
END_PROPERTY

// The month of the year extracted from the time instance.
// [get] Returns the month as an `E_Month` enum or a value ranging from 1 to 12 value.
PROPERTY Month : E_Month
GET
Month := THIS^._Date.wMonth;
END_GET
END_PROPERTY

// Updates the internal epoch milliseconds of the time instance to the current system time in UTC format.
METHOD Now : REFERENCE TO FB_TimeInstance // A reference to the current instance.
VAR_OUTPUT
	// Error code indicating the result of the operation.
	Error : FsError.T_Error;
END_VAR
VAR
	eResult : FsError.E_CodesysCmpError;
END_VAR
Now REF= THIS^;

// Get the current time instance as UTC.
eResult := SysTimeRtc.SysTimeRtcHighResGet(THIS^._nEpochMilliseconds);
CASE eResult OF
	FsError.E_CodesysCmpError.ERR_OK:
		SysTimeRtc.SysTimeRtcConvertHighResToDate(THIS^._nEpochMilliseconds, THIS^._Date);
ELSE // Reset the time instance class if there's an error.
	Error := 
		FsError.F_CreateErrorFromStartRange(
			FsError.GVL_ErrorDescriptors.fbGeneralErrorCodes,
			FsError.E_GeneralErrorCode.ERR_CODESYS_BEGIN,
			eResult);
	THIS^.FB_init(FALSE, FALSE);
	END_CASE
END_METHOD

// The second of the minute extracted from the time instance.
// [get] Returns the second component, with a value ranging from 0 to 59.
PROPERTY Second : T_Second
GET
Second := THIS^._Date.wSecond;
END_GET
END_PROPERTY

// Converts the time instance to a date value.
METHOD ToDate : DATE // The date part of the time instance.
VAR_OUTPUT
	// Error code indicating the result of the operation.
	Error : FsError.T_Error;
END_VAR
ToDate := TO_DATE(THIS^.ToDateTime(Error => Error));
END_METHOD

// Converts the time instance to a combined date and time value.
METHOD ToDateTime : DT // The combined date and time value as a DT (Date and Time).
VAR_OUTPUT
	// Error code indicating the result of the operation.
	Error : FsError.T_Error;
END_VAR
VAR
	nLocal : DWORD;
	eResult : FsError.E_CodesysCmpError;
END_VAR
CASE THIS^._eKind OF
	E_TimeInstanceKind.Local:
		eResult := SysTimeRtc.SysTimeRtcConvertUtcToLocal(
			TO_DWORD(THIS^._nEpochMilliseconds / 1000),
			nLocal);
	
		ToDateTime := TO_DT(nLocal);
		
		IF eResult <> FsError.E_CodesysCmpError.ERR_OK THEN 
			Error := 
				FsError.F_CreateErrorFromStartRange(
					FsError.GVL_ErrorDescriptors.fbGeneralErrorCodes,
					FsError.E_GeneralErrorCode.ERR_CODESYS_BEGIN,
					eResult);
			END_IF
		
ELSE 
	ToDateTime := TO_DT(THIS^._nEpochMilliseconds / 1000);
	END_CASE
END_METHOD

// Converts the time instance to local time representation.
METHOD ToLocal : I_TimeInstance // A reference to the current instance.
VAR_OUTPUT
	// Error code indicating the result of the operation.
	Error : FsError.T_Error;
END_VAR
VAR
	eResult : FsError.E_CodesysCmpError;
END_VAR
ToLocal := THIS^;

IF THIS^._eKind = E_TimeInstanceKind.Local THEN RETURN; END_IF;

eResult := SysTimeRtc.SysTimeRtcConvertHighResToLocal(THIS^._nEpochMilliseconds, THIS^._Date);
CASE eResult OF
	FsError.E_CodesysCmpError.ERR_OK:
		THIS^._eKind := E_TimeInstanceKind.Local;
ELSE
	Error := 
		FsError.F_CreateErrorFromStartRange(
			FsError.GVL_ErrorDescriptors.fbGeneralErrorCodes,
			FsError.E_GeneralErrorCode.ERR_CODESYS_BEGIN,
			eResult);
	END_CASE
END_METHOD

// Converts the time instance to a time of day  value.
METHOD ToTimeOfDay : TOD // The time of day part of the time instance.
VAR_INPUT
END_VAR
ToTimeOfDay := TO_TOD(
	(THIS^._Date.wHour * TO_DWORD(TOD#01:00:00.000))
	+
	(THIS^._Date.wMinute * TO_DWORD(TOD#00:01:00.000))
	+ 
	(THIS^._Date.wSecond * TO_DWORD(TOD#00:00:01.000))
	+ 
	THIS^._Date.wMilliseconds);
END_METHOD

// Converts the time instance to UTC time representation.
METHOD ToUTC : I_TimeInstance // A reference to the current instance.
VAR_OUTPUT
	// Error code indicating the result of the operation.
	Error : FsError.T_Error;
END_VAR
VAR
	eResult : FsError.E_CodesysCmpError;
END_VAR
ToUTC := THIS^;

IF THIS^._eKind = E_TimeInstanceKind.UTC THEN RETURN; END_IF;

eResult := SysTimeRtc.SysTimeRtcConvertHighResToDate(THIS^._nEpochMilliseconds, THIS^._Date);
CASE eResult OF
	FsError.E_CodesysCmpError.ERR_OK:
		THIS^._eKind := E_TimeInstanceKind.UTC;
ELSE
	Error := 
		FsError.F_CreateErrorFromStartRange(
			FsError.GVL_ErrorDescriptors.fbGeneralErrorCodes,
			FsError.E_GeneralErrorCode.ERR_CODESYS_BEGIN,
			eResult);
	END_CASE
END_METHOD

// The year extracted from the time instance.
// [get] Returns the year as a 4 digit value.
PROPERTY Year : T_Year
GET
Year := THIS^._Date.wYear;
END_GET
END_PROPERTY

END_FUNCTION_BLOCK

// POUs/FB_Timer
// A timing source that is used to track a specified duration. It provides methods
// to start, stop, pause, and clear the timer, and properties to track its state.
//
// [usage]
// 1. Set the desired duration using the `Duration` property.
// 2. Start the timer using the `Start` method.
// 3. Optionally, call `Pause` to pause the timer and `Start` again to resume it.
// 4. Check the `ElapsedTime` and `TimeRemaining` properties to monitor the timer’s progress.
// 5. When the timer reaches the duration, the `HasExpired` property will return `TRUE`.
{attribute 'enable_dynamic_creation'}
{attribute 'no_explicit_call' := 'direct call for this function block is not allowed'}
FUNCTION_BLOCK FINAL FB_Timer IMPLEMENTS I_Timer
VAR
    _tStartTime		: LTIME; // The time when the timer was started.
    _tPausedTime	: LTIME; // The time when the timer was paused.
    _tDuration		: LTIME; // The total duration set for the timer.
    _bIsRunning		: BOOL;  // Indicates whether the timer is currently running.
    _bHasPaused		: BOOL;  // Indicates whether the timer is currently paused.
END_VAR

// Clears the timer, resetting the elapsed time to zero.
//
// [note]
// The timer must be running for this method to take effect. If the timer is
// paused, the paused state is cleared as well.
METHOD Clear
VAR_INPUT
END_VAR
IF NOT THIS^._bIsRunning THEN RETURN; END_IF
IF THIS^._bHasPaused THEN THIS^._tPausedTime := LTIME#0S; END_IF
THIS^._tStartTime := LTIME();
END_METHOD

// The duration for the timer. It specifies how long the timer should run before
// it expires.
// [get] Returns the set duration.
// [set] Sets the duration for the timer.
PROPERTY Duration : LTIME
GET
Duration := THIS^._tDuration;
END_GET
SET
THIS^._tDuration := Duration;
END_SET
END_PROPERTY

// The elapsed time since the timer was started.
// [get] Returns the elapsed time.
PROPERTY ElapsedTime  : LTIME
GET
IF THIS^._bIsRunning THEN
	ElapsedTime :=
		SEL(THIS^._bHasPaused,
			LIMIT(LTIME#0S, LTIME() - THIS^._tStartTime, THIS^._tDuration),
			THIS^._tPausedTime);
ELSE
	ElapsedTime := LTIME#0S;
	END_IF
END_GET
END_PROPERTY

// Indicates whether the timer has expired.
// [get] Returns TRUE if the timer is running and has expired; otherwise, FALSE.
PROPERTY HasExpired : BOOL
GET
HasExpired := THIS^._bIsRunning AND (THIS^.ElapsedTime >= THIS^._tDuration);
END_GET
END_PROPERTY

// Indicates whether the timer is currently paused.
// [get] Returns TRUE if the timer is is running and paused; otherwise, FALSE.
PROPERTY HasPaused : BOOL
GET
HasPaused := THIS^._bIsRunning AND THIS^._bHasPaused;
END_GET
END_PROPERTY

// Indicates whether the timer is currently running.
// [get] Returns TRUE if the timer is running; otherwise, FALSE.
PROPERTY IsRunning  : BOOL
GET
IsRunning := THIS^._bIsRunning;
END_GET
END_PROPERTY

// Pauses the timer, preserving the elapsed time without resetting.
//
// [note]
// If the timer is already paused or not running, this method does nothing.
METHOD Pause
VAR_INPUT
END_VAR
IF (NOT THIS^._bIsRunning) OR THIS^._bHasPaused THEN RETURN; END_IF

THIS^._tPausedTime := LTIME() - THIS^._tStartTime;
THIS^._bHasPaused := TRUE;
END_METHOD

// Starts the timer, beginning the tracking of time towards the specified duration.
//
// [note]
// If the timer was previously paused, it resumes from the paused time. 
// If the timer is already running, this method does nothing.
METHOD Start
VAR_INPUT
END_VAR
IF THIS^._bIsRunning AND (NOT THIS^._bHasPaused) THEN RETURN; END_IF

THIS^._tStartTime :=
	SEL(THIS^._bHasPaused, LTIME(), LTIME() - THIS^._tPausedTime);

THIS^._bIsRunning := TRUE;
THIS^._bHasPaused := FALSE;
END_METHOD

// Stops the timer, halting the tracking of time.
//
//[note]
// If the timer is not running, this method does nothing.
// If the timer is paused it's pause state will be cleared.
METHOD Stop
VAR_INPUT
END_VAR
IF NOT THIS^._bIsRunning THEN RETURN; END_IF

THIS^._bIsRunning := FALSE;
THIS^._bHasPaused := FALSE;
END_METHOD

// The remaining time until the timer expires.
// [get] Returns the time remaining until expiration.
PROPERTY TimeRemaining : LTIME
GET
VAR
	tElapsedTime : LTIME;
END_VAR
tElapsedTime := THIS^.ElapsedTime;
TimeRemaining := MAX(THIS^._tDuration, tElapsedTime) - tElapsedTime;
END_GET
END_PROPERTY

END_FUNCTION_BLOCK

// POUs/FB_TimeSpan
// A function block that represents a time span, providing properties and methods
// to manipulate and convert time durations.
// It implements interfaces for time span operations and properties.
//
// [usage]
// 1. Use `FromTime` or `FromShortTime` methods to initialise the time span.
// 2. Access properties like `Days`, `Hours`, `Minutes`, etc., to retrieve specific
//    components of the time span.
// 3. Utilise conversion methods like `ToSeconds`, `ToMilliseconds`, etc., to get
//    the duration in different time units.
{attribute 'enable_dynamic_creation'}
{attribute 'no_explicit_call' := 'direct call for this function block is not allowed'}
FUNCTION_BLOCK FINAL FB_TimeSpan 
IMPLEMENTS 
	I_TimeSpan, I_TimeSpanProperties, I_TimeSpanConversions
VAR
	_tTick : LTIME; // Stores the time duration in LTIME format.
END_VAR

// The day component of the time span.
// [get] Returns the day component of the time, with a value ranging from 0 to 213503.
PROPERTY Day : UDINT(0..213503)
GET
Day := TO_UDINT(TO_ULINT(THIS^._tTick) / TO_ULINT(LTIME#1D));
END_GET
END_PROPERTY

// Sets the time span based on the given `TIME` value.
// Initialises the time span using an `TIME` value.
//
// [Note]
// `TIME` has a lower precision compared to `LTIME`.
METHOD FromShortTime : I_TimeSpan // A reference to the current instance.
VAR_INPUT
	// The value used to set the time span.
	tValue : TIME;
END_VAR
FromShortTime := THIS^;

THIS^._tTick := TO_LTIME(tValue);
END_METHOD

// Sets the time span based on the given `LTIME` value.
// Initialises the time span using an `LTIME` value, which can represent time durations with high precision.
METHOD FromTime : I_TimeSpan // A reference to the current instance.
VAR_INPUT
	// The value used to set the time span.
	tValue : LTIME;
END_VAR
FromTime := THIS^;

THIS^._tTick := tValue;
END_METHOD

// The hour component of the time span.
// [get] Returns the hour component of the time, with a value ranging from 0 to 23.
PROPERTY Hour : T_Hour
GET
Hour := 
	TO_UINT(
		(
			TO_ULINT(THIS^._tTick) MOD TO_ULINT(LTIME#1D)
		)
		/ TO_ULINT(LTIME#1H));
END_GET
END_PROPERTY

// The microsecond component of the time span.
// [get] Returns the microsecond component, with a value ranging from 0 to 999.
PROPERTY Microsecond : T_Microsecond
GET
Microsecond := 
	TO_UINT(
		(
			TO_ULINT(THIS^._tTick) MOD TO_ULINT(LTIME#1MS)
		)
		/ TO_ULINT(LTIME#1US));
END_GET
END_PROPERTY

// The millisecond component of the time span.
// [get] Returns the millisecond component, with a value ranging from 0 to 999.
PROPERTY Millisecond : T_Millisecond
GET
Millisecond := 
	TO_UINT(
		(
			TO_ULINT(THIS^._tTick) MOD TO_ULINT(LTIME#1S)
		)
		/ TO_ULINT(LTIME#1MS));
END_GET
END_PROPERTY

// The minute component of the time span.
// [get] Returns the minute component, with a value ranging from 0 to 59.
PROPERTY Minute : T_Minute
GET
Minute :=
	TO_UINT(
		(
			TO_ULINT(THIS^._tTick) MOD TO_ULINT(LTIME#1H)
		) 
		/ TO_ULINT(LTIME#1M));
END_GET
END_PROPERTY

// The nanosecond component of the time span.
// [get] Returns the nanosecond component, with a value ranging from 0 to 999.
PROPERTY Nanosecond : T_Nanosecond
GET
Nanosecond := 
	TO_UINT(
		(
			TO_ULINT(THIS^._tTick) MOD TO_ULINT(LTIME#1US)
		)
		/ TO_ULINT(LTIME#1NS));
END_GET
END_PROPERTY

// Sets the time span to the system's tick value.
METHOD Now : I_TimeSpan // A reference to the current time span instance.
VAR_INPUT
END_VAR
Now := THIS^;

THIS^._tTick := LTIME();
END_METHOD

// The second component of the time span.
// [get] Returns the second component, with a value ranging from 0 to 59.
PROPERTY Second : T_Second
GET
Second := 
	TO_UINT(
		(
			TO_ULINT(THIS^._tTick) MOD TO_ULINT(TIME#1M)
		) 
		/ TO_ULINT(LTIME#1S));
END_GET
END_PROPERTY

// The reference to the current time span.
// [get] Returns a reference to the current time instance implementing `I_TimeSpan`.
PROPERTY Span : I_TimeSpan
GET
Span := THIS^;
END_GET
END_PROPERTY

// Represents the time span as LTIME.
// [get] Returns the time span value as an LTIME, which can be used for time calculations and comparisons.
PROPERTY Tick : LTIME
GET
Tick := THIS^._tTick;
END_GET
END_PROPERTY

// Converts the time span represented by the instance into days.
METHOD ToDays : ULINT // The total number of days in the time span.
VAR_INPUT
END_VAR
ToDays := TO_ULINT(THIS^._tTick) / TO_ULINT(LTIME#1D);
END_METHOD

// Converts the time span represented by the instance into hours.
METHOD ToHours : ULINT // The total number of hours in the time span.
VAR_INPUT
END_VAR
ToHours := TO_ULINT(THIS^._tTick) / TO_ULINT(LTIME#1H);
END_METHOD

// Converts the time span represented by the instance into microseconds.
METHOD ToMicroseconds : ULINT // The total number of microseconds in the time span.
VAR_INPUT
END_VAR
ToMicroseconds := TO_ULINT(THIS^._tTick) / TO_ULINT(LTIME#1US);
END_METHOD

// Converts the time span represented by the instance into milliseconds.
METHOD ToMilliseconds : ULINT // The total number of milliseconds in the time span.
VAR_INPUT
END_VAR
ToMilliseconds := TO_ULINT(THIS^._tTick) / TO_ULINT(LTIME#1MS);
END_METHOD

// Converts the time span represented by the instance into minutes.
METHOD ToMinutes : ULINT // The total number of minutes in the time span.
VAR_INPUT
END_VAR
ToMinutes := TO_ULINT(THIS^._tTick) / TO_ULINT(LTIME#1M);
END_METHOD

// Converts the time span represented by the instance into nanoseconds.
METHOD ToNanoseconds : ULINT // The total number of nanoseconds in the time span.
VAR_INPUT
END_VAR
ToNanoseconds := TO_ULINT(THIS^._tTick);
END_METHOD

// Converts the time span represented by the instance into seconds.
METHOD ToSeconds : ULINT // The total number of seconds in the time span.
VAR_INPUT
END_VAR
ToSeconds := TO_ULINT(THIS^._tTick) / TO_ULINT(LTIME#1S);
END_METHOD

END_FUNCTION_BLOCK

// POUs/PLAYGROUND
{attribute 'no_explicit_call' := 'direct call for this program is not allowed'} 
PROGRAM INTERNAL PLAYGROUND
VAR
	bStart,
	bStop,
	bPause,
	bClear 			: BOOL;
	eKind			: E_TimeInstanceKind := E_TimeInstanceKind.Local;
	nValue 			: ULINT;
	tValue,
	tValue2			: LTIME	;
	tSetpoint 		: LTIME := LTIME#10S;
	dTimestamp 		: DATE;
	dtTimestamp 	: DT;
	tdTimestamp 	: TOD;
	eDay 			: E_DayOfWeek;
	eMonth 			: E_Month;
	Count 			: FsCommon.T_Size;
	fbIntervalTimer : FB_IntervalTimer;
	fbStopwatch 	: FB_Stopwatch;
	fbTimer 		: FB_Timer;
	fbTimestamp 	: FB_TimeInstance;
	fbTimeSpan		: FB_TimeSpan;
END_VAR

Example1();
nValue := fbTimeSpan.FromTime(LTIME#100D2H30M40S500MS600US700NS).ToMinutes();
(*
fbTimestamp.Now(Error => );

CASE eKind OF
	E_TimeInstanceKind.UTC:
		fbTimestamp.ToUTC(Error =>);
		
	E_TimeInstanceKind.Local:
		fbTimestamp.ToLocal(Error =>);
	END_CASE
	
dTimestamp	:= fbTimestamp.ToDate();
dtTimestamp := fbTimestamp.ToDateTime();
tdTimestamp := fbTimestamp.ToTimeOfDay();
eDay 		:= fbTimestamp.DayOfWeek;
eMonth 		:= fbTimestamp.Month;
*)
(*

*)
(*
IF FsCommon.F_ResetOnTrue(bStart) THEN fbTimer.Start(); END_IF
IF FsCommon.F_ResetOnTrue(bStop)  THEN fbTimer.Stop(); 	END_IF
IF FsCommon.F_ResetOnTrue(bPause) THEN fbTimer.Pause(); END_IF
IF FsCommon.F_ResetOnTrue(bClear) THEN fbTimer.Clear(); END_IF

fbTimer.Duration := tSetpoint;
tValue	:= fbTimer.ElapsedTime;
tValue2 := fbTimer.TimeRemaining;
*)
(*
fbIntervalTimer.IntervalTime := LTIME#10S;

tValue := 
	fbIntervalTimer
		.SetCallback(0)
		.Start()
		.Run()
		.ElapsedTime;
		
Count := fbIntervalTimer.IntervalCount;
*)

METHOD Example1
VAR_STAT
	sValue 			: Tc2_System.T_MaxString;
	dtTimestamp		: DT;
	fbTimestamp 	: FB_TimeInstance;
	bCreate			: BOOL := TRUE;
	Err             : FsError.T_Error;
    fbWithAdsLogger : FsError.FB_AdsErrorLogger;
END_VAR
IF FsCommon.F_ResetOnTrue(bCreate) THEN
	dtTimestamp := fbTimestamp.Now(Error => Err).ToLocal().ToDateTime();
	
	IF Err.IsRaised THEN Err.LogMessage(fbWithAdsLogger); RETURN; END_IF
	
	sValue := '';
	sValue := Tc2_Standard.CONCAT('Today is ', TO_STRING(fbTimestamp.DayOfWeek));
	sValue := Tc2_Standard.CONCAT(sValue, ', ');
	sValue := Tc2_Standard.CONCAT(sValue, TO_STRING(fbTimestamp.DayOfMonth));
	sValue := Tc2_Standard.CONCAT(sValue, ' ');
	sValue := Tc2_Standard.CONCAT(sValue, TO_STRING(fbTimestamp.Month));
	sValue := Tc2_Standard.CONCAT(sValue, ' ');
	sValue := Tc2_Standard.CONCAT(sValue, TO_STRING(fbTimestamp.Year));
	sValue := Tc2_Standard.CONCAT(sValue, '.');
	END_IF
END_METHOD

END_PROGRAM

// Project Information/F_GetCompany
// This function has been automatically generated from the project information.
{attribute 'signature_flag' := '1073741824'}
{attribute 'TcGenerated'}
{attribute 'no-analysis'}
FUNCTION F_GetCompany : WSTRING
VAR_INPUT
	
END_VAR

F_GetCompany := "FisoThemes";

END_FUNCTION

// Project Information/F_GetTitle
// This function has been automatically generated from the project information.
{attribute 'signature_flag' := '1073741824'}
{attribute 'TcGenerated'}
{attribute 'no-analysis'}
FUNCTION F_GetTitle : WSTRING
VAR_INPUT
	
END_VAR

F_GetTitle := "FsTime";

END_FUNCTION

// Project Information/F_GetVersion
// This function has been automatically generated from the project information.
{attribute 'signature_flag' := '1073741824'}
{attribute 'TcGenerated'}
{attribute 'no-analysis'}
FUNCTION F_GetVersion : ST_LibVersion
VAR_INPUT
	
END_VAR

F_GetVersion.iMajor := 0;
F_GetVersion.iMinor := 1;
F_GetVersion.iBuild := 0;
F_GetVersion.iRevision := 0;

END_FUNCTION
